// TIA Portal V18 export
DATA_BLOCK "MOT2_remSel"   // DB19
VERSION : 0.1
// stored: AutoNumber true, DBAccessibleFromOPCUA true, InstanceOfName axis_manager, InstanceOfType FB
"axis_manager"
   // VAR_INPUT
   //    allowed : Bool;
   //    targetUnison : Real;
   //    targetHome : Real;
   //    targetStep : Real;
   //    bSoftStop : Bool;
   //    bHome : Bool;
   //    hbStepPlus : Bool;
   //    hbStepMinus : Bool;
   //    bFwd : Bool;
   //    bRev : Bool;
   //    Params : "typeMotPara";
   //    ExecUni : Bool;
   //    theseAreDoors : Bool;
   //    xOverrideLOCAL : Bool;
   //    POS : Real;
   // END_VAR
   // VAR_OUTPUT
   //    team_unison : Bool;
   //    team_free : Bool;
   //    team_override : Bool;
   //    Desk_slowly : Bool;
   //    yaSpeedManual : Real;
   //    yaSpeedAuto : Real;
   //    m_auto : Bool;
   //    m_man : Bool;
   //    au_execute : Bool;
   //    aut_target : Real;
   //    OVERRIDE : Bool;
   //    ExecutingManuverFreeMode : Bool;
   // END_VAR
   // VAR
   //    st_Fwd : Bool;
   //    st_Rev : Bool;
   //    st_speed_slow_or_fast_negative : Real;
   //    aman_sel_target_Instance { S7_SetPoint := 'True'} : "aman_sel_target";
   // END_VAR
BEGIN
END_DATA_BLOCK
